TYPE ST_PNOutput_OutputField:
STRUCT
	w_Status					:	WORD;
	w_Warnings					:	WORD;
	w_Faults					:	WORD;
	i_ActivePower				:	INT;
	i_ReactivePower				:	INT;
	i_PowerFactor				:	INT;
	ui_Frequency				:	UINT;
	ui_VoltageL1N				:	UINT;
	ui_VoltageL2N				:	UINT;
	ui_VoltageL3N				:	UINT;
	ui_VoltageL1L2				:	UINT;
	ui_VoltageL2L3				:	UINT;
	ui_VoltageL3L1				:	UINT;
	ui_CurrentL1				:	UINT;
	ui_CurrentL2				:	UINT;
	ui_CurrentL3				:	UINT;
	ui_CurrentN					:	UINT;
	ui_CurrentLimitField		:	UINT;
	udi_TotalEnergySupplied 	:	UDINT;
	udi_TotalEnergyConsumed 	:	UDINT;
	ui_Current1L1				:	UINT;
	ui_Current1L2				:	UINT;
	ui_Current1L3				:	UINT;
	ui_Current1N				:	UINT;
	ui_Current2L1				:	UINT;
	ui_Current2L2				:	UINT;
	ui_Current2L3				:	UINT;
	ui_Current2N				:	UINT;
	ui_Current3L1				:	UINT;
	ui_Current3L2				:	UINT;
	ui_Current3L3				:	UINT;
	ui_Current3N				:	UINT;
END_STRUCT
END_TYPE

(* stored: Version 1.1.0.1, ProductVersion 3.1.4026.18
   DUT ST_PNOutput_OutputField: Id {049f9c24-aeb2-49bc-8a5b-b602605bfa85} *)
